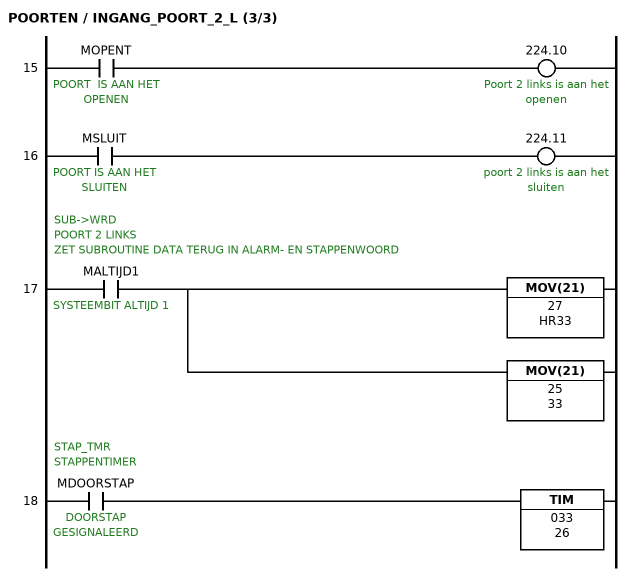
; [picture p445: POORTEN / INGANG_POORT_2_L, rungs 15-18]
; rung 15
LD MOPENT  ; POORT  IS AAN HET OPENEN
OUT 224.10  ; Poort 2 links is aan het openen
; rung 16
LD MSLUIT  ; POORT IS AAN HET SLUITEN
OUT 224.11  ; poort 2 links is aan het sluiten
; rung 17: SUB->WRD / POORT 2 LINKS / ZET SUBROUTINE DATA TERUG IN ALARM- EN STAPPENWOORD
LD MALTIJD1  ; SYSTEEMBIT ALTIJD 1
MOV(21) 27 HR33
MOV(21) 25 33
; rung 18: STAP_TMR / STAPPENTIMER
LD MDOORSTAP  ; DOORSTAP GESIGNALEERD
TIM 033 26

### Section INGANG_POORT_2_R

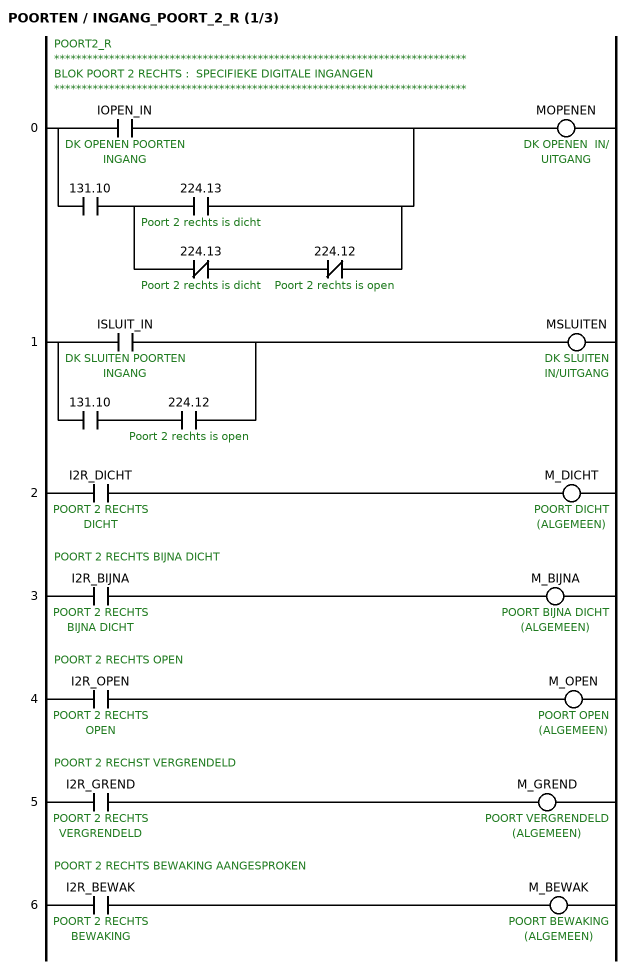
; rung 0: POORT2_R / *************************************************************************** / BLOK POORT 2 RECHTS :  SPECIFIEKE DIGITALE INGANGEN / ***************************************************************************
LD IOPEN_IN  ; DK OPENEN POORTEN INGANG
LD 131.10
LD 224.13  ; Poort 2 rechts is dicht
LDNOT 224.13  ; Poort 2 rechts is dicht
ANDNOT 224.12  ; Poort 2 rechts is open
ORLD
ANDLD
ORLD
OUT MOPENEN  ; DK OPENEN  IN/ UITGANG
; rung 1
LD ISLUIT_IN  ; DK SLUITEN POORTEN INGANG
LD 131.10
AND 224.12  ; Poort 2 rechts is open
ORLD
OUT MSLUITEN  ; DK SLUITEN  IN/UITGANG
; rung 2
LD I2R_DICHT  ; POORT 2 RECHTS DICHT
OUT M_DICHT  ; POORT DICHT (ALGEMEEN)
; rung 3: POORT 2 RECHTS BIJNA DICHT
LD I2R_BIJNA  ; POORT 2 RECHTS BIJNA DICHT
OUT M_BIJNA  ; POORT BIJNA DICHT  (ALGEMEEN)
; rung 4: POORT 2 RECHTS OPEN
LD I2R_OPEN  ; POORT 2 RECHTS OPEN
OUT M_OPEN  ; POORT OPEN (ALGEMEEN)
; rung 5: POORT 2 RECHST VERGRENDELD
LD I2R_GREND  ; POORT 2 RECHTS VERGRENDELD
OUT M_GREND  ; POORT VERGRENDELD (ALGEMEEN)
; rung 6: POORT 2 RECHTS BEWAKING AANGESPROKEN
LD I2R_BEWAK  ; POORT 2 RECHTS BEWAKING
OUT M_BEWAK  ; POORT BEWAKING (ALGEMEEN)

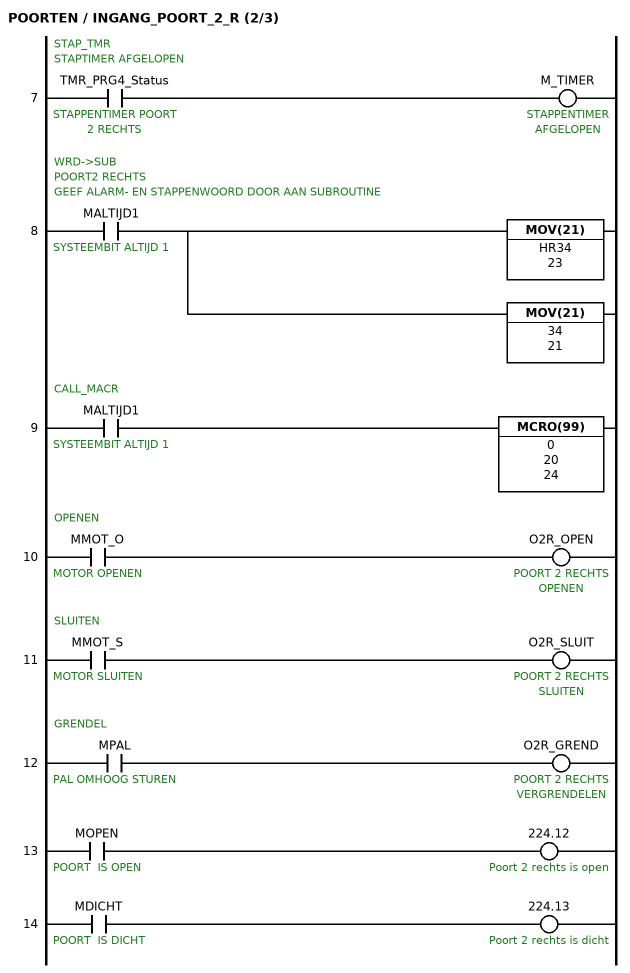
; rung 7: STAP_TMR / STAPTIMER AFGELOPEN
LD TMR_PRG4_Status  ; STAPPENTIMER POORT 2 RECHTS
OUT M_TIMER  ; STAPPENTIMER AFGELOPEN
; rung 8: WRD->SUB / POORT2 RECHTS / GEEF ALARM- EN STAPPENWOORD DOOR AAN SUBROUTINE
LD MALTIJD1  ; SYSTEEMBIT ALTIJD 1
MOV(21) HR34 23
MOV(21) 34 21
; rung 9: CALL_MACR
LD MALTIJD1  ; SYSTEEMBIT ALTIJD 1
MCRO(99) 0 20 24
; rung 10: OPENEN
LD MMOT_O  ; MOTOR OPENEN
OUT O2R_OPEN  ; POORT 2 RECHTS OPENEN
; rung 11: SLUITEN
LD MMOT_S  ; MOTOR SLUITEN
OUT O2R_SLUIT  ; POORT 2 RECHTS SLUITEN
; rung 12: GRENDEL
LD MPAL  ; PAL OMHOOG STUREN
OUT O2R_GREND  ; POORT 2 RECHTS VERGRENDELEN
; rung 13
LD MOPEN  ; POORT  IS OPEN
OUT 224.12  ; Poort 2 rechts is open
; rung 14
LD MDICHT  ; POORT  IS DICHT
OUT 224.13  ; Poort 2 rechts is dicht

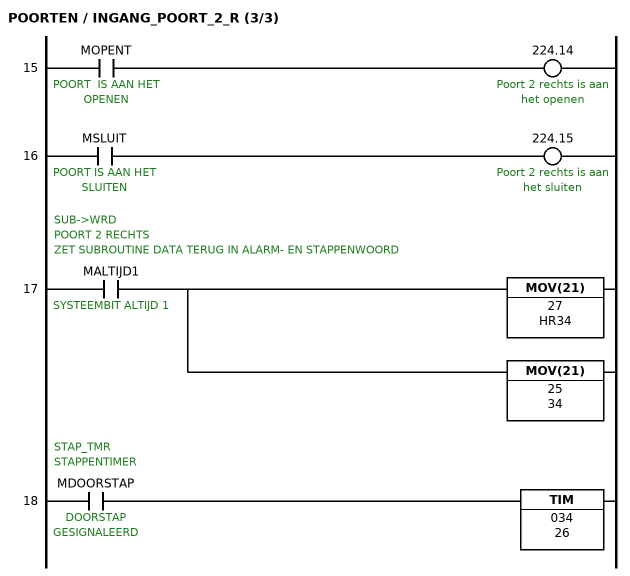
; rung 15
LD MOPENT  ; POORT  IS AAN HET OPENEN
OUT 224.14  ; Poort 2 rechts is aan het openen
; rung 16
LD MSLUIT  ; POORT IS AAN HET SLUITEN
OUT 224.15  ; Poort 2 rechts is aan het sluiten
; rung 17: SUB->WRD / POORT 2 RECHTS / ZET SUBROUTINE DATA TERUG IN ALARM- EN STAPPENWOORD
LD MALTIJD1  ; SYSTEEMBIT ALTIJD 1
MOV(21) 27 HR34
MOV(21) 25 34
; rung 18: STAP_TMR / STAPPENTIMER
LD MDOORSTAP  ; DOORSTAP GESIGNALEERD
TIM 034 26

### Section UITGANG_POORT_3_L

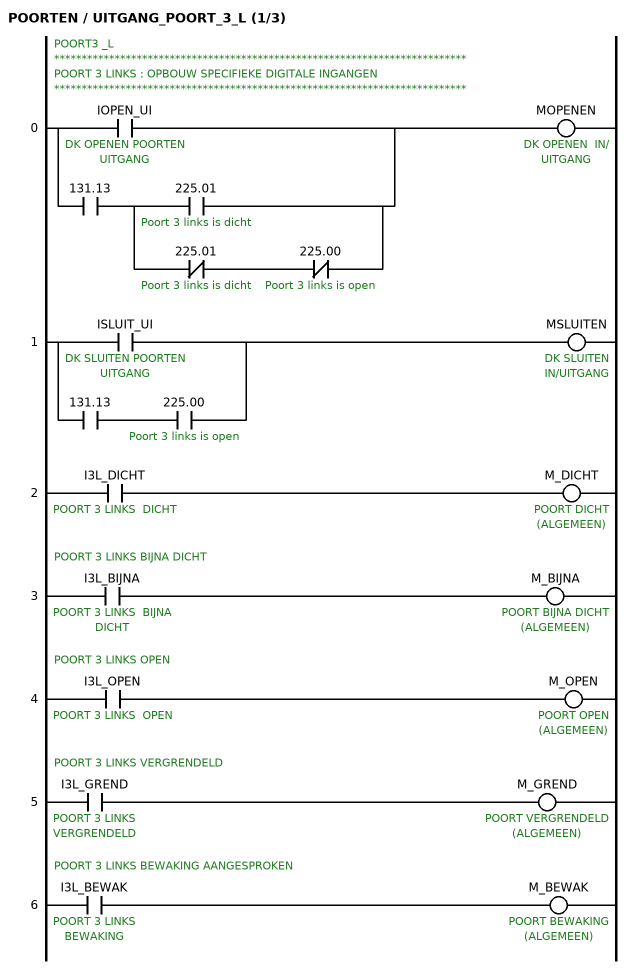
; rung 0: POORT3 _L / *************************************************************************** / POORT 3 LINKS : OPBOUW SPECIFIEKE DIGITALE INGANGEN / ***************************************************************************
LD IOPEN_UI  ; DK OPENEN POORTEN UITGANG
LD 131.13
LD 225.01  ; Poort 3 links is dicht
LDNOT 225.01  ; Poort 3 links is dicht
ANDNOT 225.00  ; Poort 3 links is open
ORLD
ANDLD
ORLD
OUT MOPENEN  ; DK OPENEN  IN/ UITGANG
; rung 1
LD ISLUIT_UI  ; DK SLUITEN POORTEN UITGANG
LD 131.13
AND 225.00  ; Poort 3 links is open
ORLD
OUT MSLUITEN  ; DK SLUITEN  IN/UITGANG
; rung 2
LD I3L_DICHT  ; POORT 3 LINKS  DICHT
OUT M_DICHT  ; POORT DICHT (ALGEMEEN)
; rung 3: POORT 3 LINKS BIJNA DICHT
LD I3L_BIJNA  ; POORT 3 LINKS  BIJNA DICHT
OUT M_BIJNA  ; POORT BIJNA DICHT  (ALGEMEEN)
; rung 4: POORT 3 LINKS OPEN
LD I3L_OPEN  ; POORT 3 LINKS  OPEN
OUT M_OPEN  ; POORT OPEN (ALGEMEEN)
; rung 5: POORT 3 LINKS VERGRENDELD
LD I3L_GREND  ; POORT 3 LINKS VERGRENDELD
OUT M_GREND  ; POORT VERGRENDELD (ALGEMEEN)
; rung 6: POORT 3 LINKS BEWAKING AANGESPROKEN
LD I3L_BEWAK  ; POORT 3 LINKS BEWAKING
OUT M_BEWAK  ; POORT BEWAKING (ALGEMEEN)

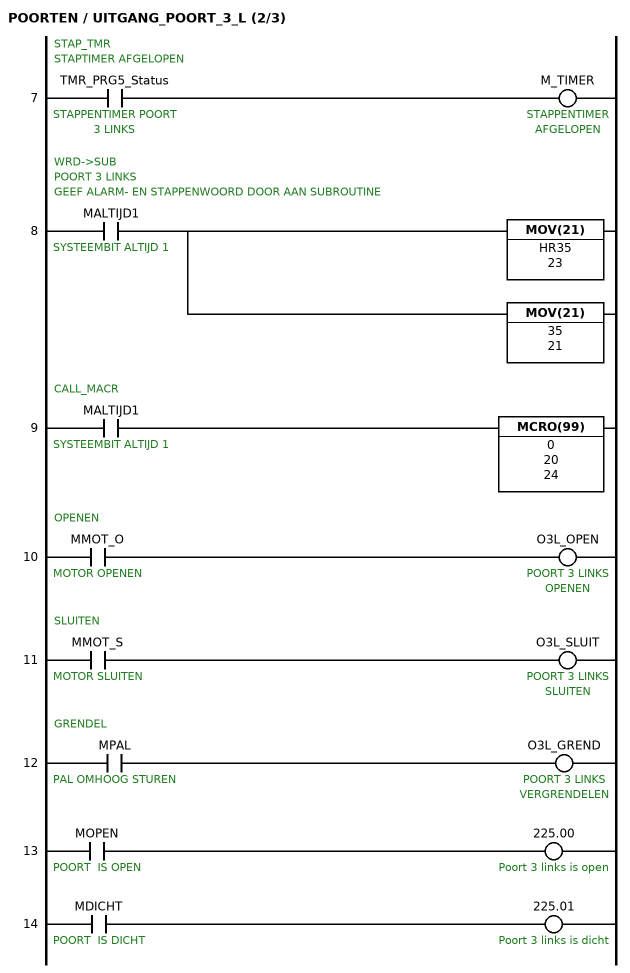
; rung 7: STAP_TMR / STAPTIMER AFGELOPEN
LD TMR_PRG5_Status  ; STAPPENTIMER POORT 3 LINKS
OUT M_TIMER  ; STAPPENTIMER AFGELOPEN
; rung 8: WRD->SUB / POORT 3 LINKS / GEEF ALARM- EN STAPPENWOORD DOOR AAN SUBROUTINE
LD MALTIJD1  ; SYSTEEMBIT ALTIJD 1
MOV(21) HR35 23
MOV(21) 35 21
; rung 9: CALL_MACR
LD MALTIJD1  ; SYSTEEMBIT ALTIJD 1
MCRO(99) 0 20 24
; rung 10: OPENEN
LD MMOT_O  ; MOTOR OPENEN
OUT O3L_OPEN  ; POORT 3 LINKS OPENEN
; rung 11: SLUITEN
LD MMOT_S  ; MOTOR SLUITEN
OUT O3L_SLUIT  ; POORT 3 LINKS SLUITEN
; rung 12: GRENDEL
LD MPAL  ; PAL OMHOOG STUREN
OUT O3L_GREND  ; POORT 3 LINKS VERGRENDELEN
; rung 13
LD MOPEN  ; POORT  IS OPEN
OUT 225.00  ; Poort 3 links is open
; rung 14
LD MDICHT  ; POORT  IS DICHT
OUT 225.01  ; Poort 3 links is dicht

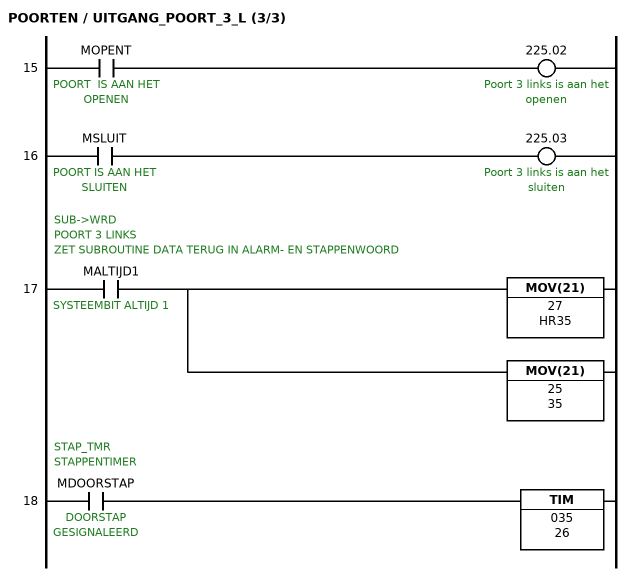
; rung 15
LD MOPENT  ; POORT  IS AAN HET OPENEN
OUT 225.02  ; Poort 3 links is aan het openen
; rung 16
LD MSLUIT  ; POORT IS AAN HET SLUITEN
OUT 225.03  ; Poort 3 links is aan het sluiten
; rung 17: SUB->WRD / POORT 3 LINKS / ZET SUBROUTINE DATA TERUG IN ALARM- EN STAPPENWOORD
LD MALTIJD1  ; SYSTEEMBIT ALTIJD 1
MOV(21) 27 HR35
MOV(21) 25 35
; rung 18: STAP_TMR / STAPPENTIMER
LD MDOORSTAP  ; DOORSTAP GESIGNALEERD
TIM 035 26

### Section UITGANG_POORT_3_R

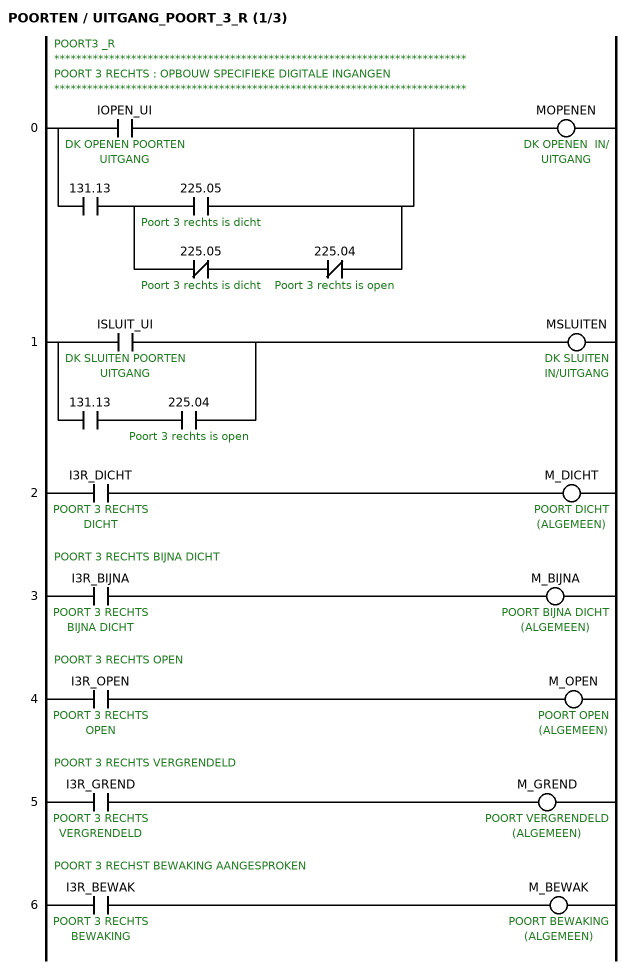
; rung 0: POORT3 _R / *************************************************************************** / POORT 3 RECHTS : OPBOUW SPECIFIEKE DIGITALE INGANGEN / ***************************************************************************
LD IOPEN_UI  ; DK OPENEN POORTEN UITGANG
LD 131.13
LD 225.05  ; Poort 3 rechts is dicht
LDNOT 225.05  ; Poort 3 rechts is dicht
ANDNOT 225.04  ; Poort 3 rechts is open
ORLD
ANDLD
ORLD
OUT MOPENEN  ; DK OPENEN  IN/ UITGANG
; rung 1
LD ISLUIT_UI  ; DK SLUITEN POORTEN UITGANG
LD 131.13
AND 225.04  ; Poort 3 rechts is open
ORLD
OUT MSLUITEN  ; DK SLUITEN  IN/UITGANG
; rung 2
LD I3R_DICHT  ; POORT 3 RECHTS DICHT
OUT M_DICHT  ; POORT DICHT (ALGEMEEN)
; rung 3: POORT 3 RECHTS BIJNA DICHT
LD I3R_BIJNA  ; POORT 3 RECHTS BIJNA DICHT
OUT M_BIJNA  ; POORT BIJNA DICHT  (ALGEMEEN)
; rung 4: POORT 3 RECHTS OPEN
LD I3R_OPEN  ; POORT 3 RECHTS OPEN
OUT M_OPEN  ; POORT OPEN (ALGEMEEN)
; rung 5: POORT 3 RECHTS VERGRENDELD
LD I3R_GREND  ; POORT 3 RECHTS VERGRENDELD
OUT M_GREND  ; POORT VERGRENDELD (ALGEMEEN)
; rung 6: POORT 3 RECHST BEWAKING AANGESPROKEN
LD I3R_BEWAK  ; POORT 3 RECHTS BEWAKING
OUT M_BEWAK  ; POORT BEWAKING (ALGEMEEN)

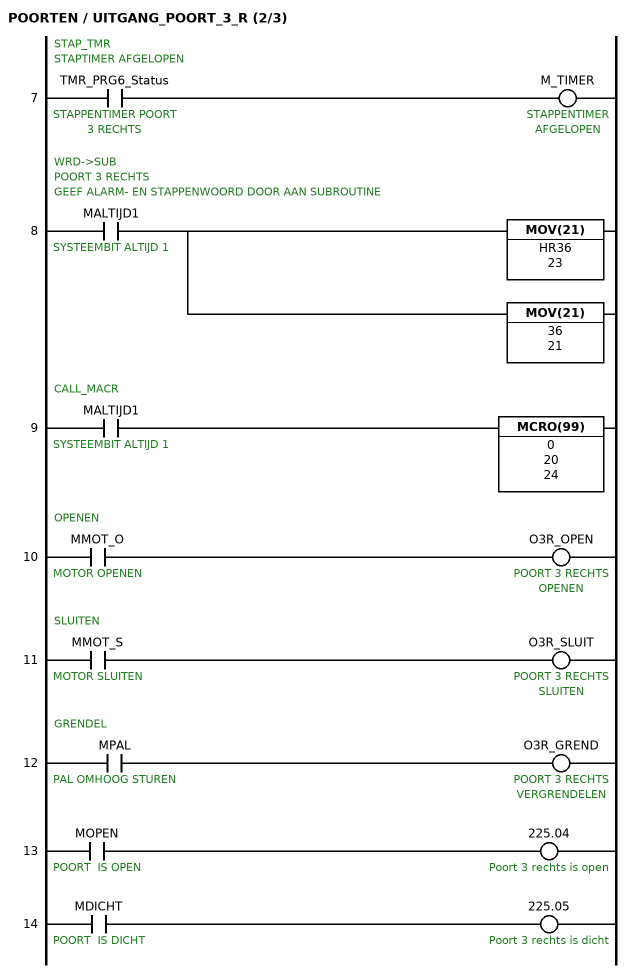
; rung 7: STAP_TMR / STAPTIMER AFGELOPEN
LD TMR_PRG6_Status  ; STAPPENTIMER POORT 3 RECHTS
OUT M_TIMER  ; STAPPENTIMER AFGELOPEN
; rung 8: WRD->SUB / POORT 3 RECHTS / GEEF ALARM- EN STAPPENWOORD DOOR AAN SUBROUTINE
LD MALTIJD1  ; SYSTEEMBIT ALTIJD 1
MOV(21) HR36 23
MOV(21) 36 21
; rung 9: CALL_MACR
LD MALTIJD1  ; SYSTEEMBIT ALTIJD 1
MCRO(99) 0 20 24
; rung 10: OPENEN
LD MMOT_O  ; MOTOR OPENEN
OUT O3R_OPEN  ; POORT 3 RECHTS OPENEN
; rung 11: SLUITEN
LD MMOT_S  ; MOTOR SLUITEN
OUT O3R_SLUIT  ; POORT 3 RECHTS SLUITEN
; rung 12: GRENDEL
LD MPAL  ; PAL OMHOOG STUREN
OUT O3R_GREND  ; POORT 3 RECHTS VERGRENDELEN
; rung 13
LD MOPEN  ; POORT  IS OPEN
OUT 225.04  ; Poort 3 rechts is open
; rung 14
LD MDICHT  ; POORT  IS DICHT
OUT 225.05  ; Poort 3 rechts is dicht

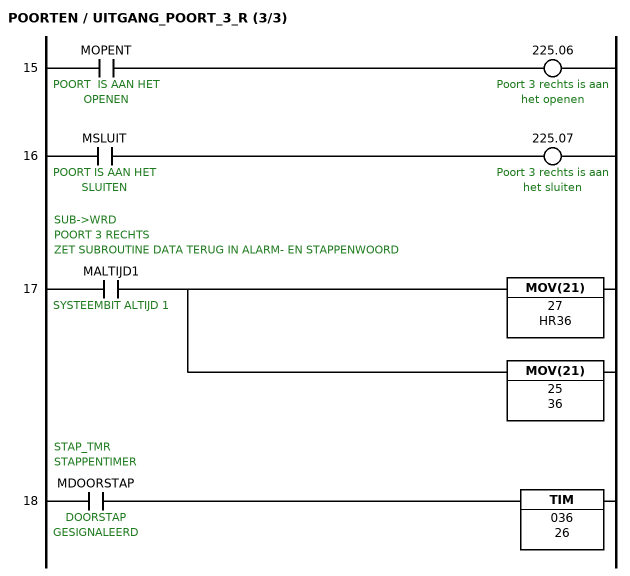
; rung 15
LD MOPENT  ; POORT  IS AAN HET OPENEN
OUT 225.06  ; Poort 3 rechts is aan het openen
; rung 16
LD MSLUIT  ; POORT IS AAN HET SLUITEN
OUT 225.07  ; Poort 3 rechts is aan het sluiten
; rung 17: SUB->WRD / POORT 3 RECHTS / ZET SUBROUTINE DATA TERUG IN ALARM- EN STAPPENWOORD
LD MALTIJD1  ; SYSTEEMBIT ALTIJD 1
MOV(21) 27 HR36
MOV(21) 25 36
; rung 18: STAP_TMR / STAPPENTIMER
LD MDOORSTAP  ; DOORSTAP GESIGNALEERD
TIM 036 26

### Section UITGANG_POORT_4_L

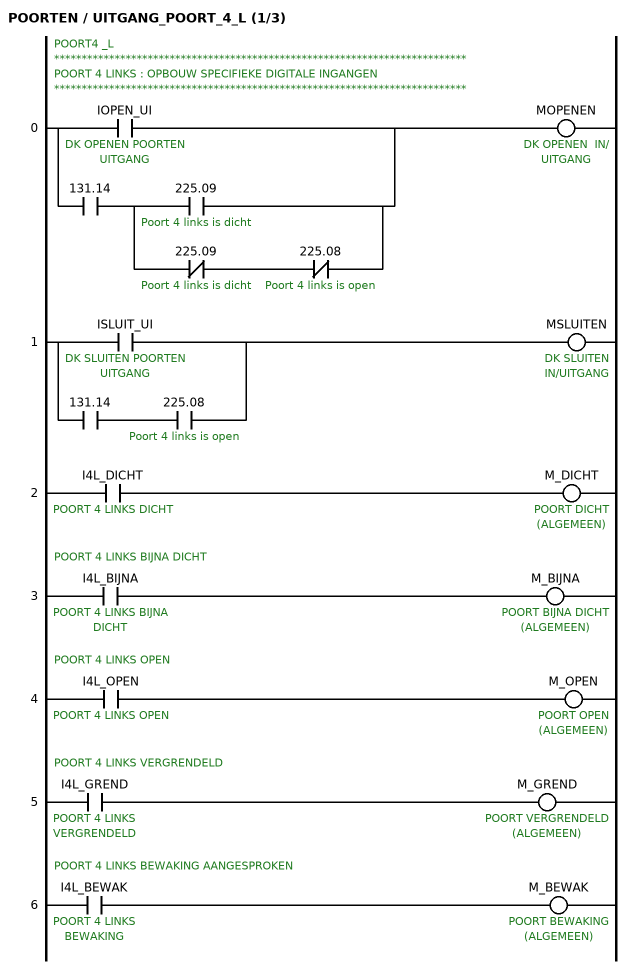
; rung 0: POORT4 _L / *************************************************************************** / POORT 4 LINKS : OPBOUW SPECIFIEKE DIGITALE INGANGEN / ***************************************************************************
LD IOPEN_UI  ; DK OPENEN POORTEN UITGANG
LD 131.14
LD 225.09  ; Poort 4 links is dicht
LDNOT 225.09  ; Poort 4 links is dicht
ANDNOT 225.08  ; Poort 4 links is open
ORLD
ANDLD
ORLD
OUT MOPENEN  ; DK OPENEN  IN/ UITGANG
; rung 1
LD ISLUIT_UI  ; DK SLUITEN POORTEN UITGANG
LD 131.14
AND 225.08  ; Poort 4 links is open
ORLD
OUT MSLUITEN  ; DK SLUITEN  IN/UITGANG
; rung 2
LD I4L_DICHT  ; POORT 4 LINKS DICHT
OUT M_DICHT  ; POORT DICHT (ALGEMEEN)
; rung 3: POORT 4 LINKS BIJNA DICHT
LD I4L_BIJNA  ; POORT 4 LINKS BIJNA DICHT
OUT M_BIJNA  ; POORT BIJNA DICHT  (ALGEMEEN)
; rung 4: POORT 4 LINKS OPEN
LD I4L_OPEN  ; POORT 4 LINKS OPEN
OUT M_OPEN  ; POORT OPEN (ALGEMEEN)
; rung 5: POORT 4 LINKS VERGRENDELD
LD I4L_GREND  ; POORT 4 LINKS VERGRENDELD
OUT M_GREND  ; POORT VERGRENDELD (ALGEMEEN)
; rung 6: POORT 4 LINKS BEWAKING AANGESPROKEN
LD I4L_BEWAK  ; POORT 4 LINKS BEWAKING
OUT M_BEWAK  ; POORT BEWAKING (ALGEMEEN)

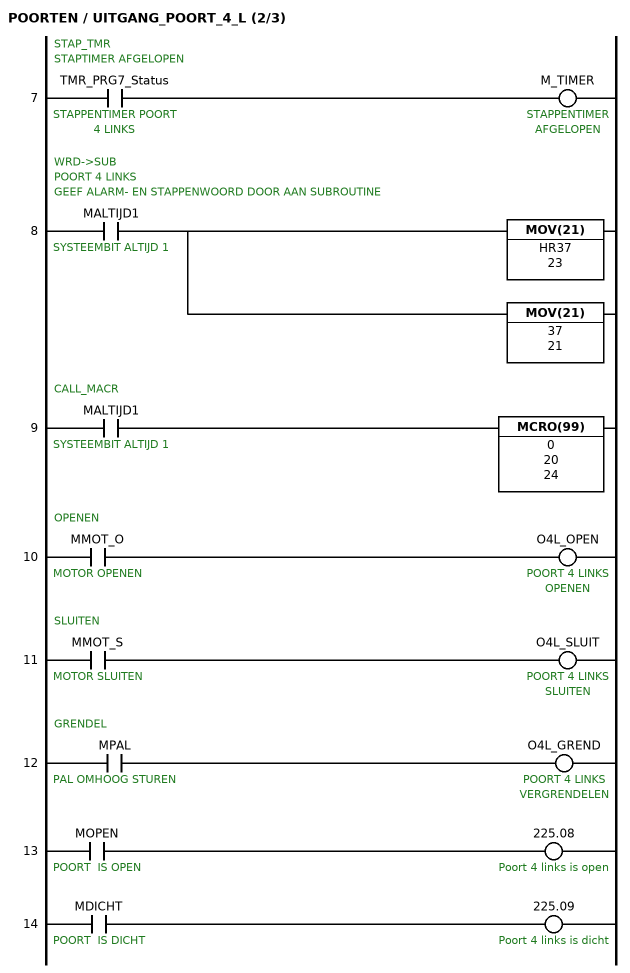
; rung 7: STAP_TMR / STAPTIMER AFGELOPEN
LD TMR_PRG7_Status  ; STAPPENTIMER POORT 4 LINKS
OUT M_TIMER  ; STAPPENTIMER AFGELOPEN
; rung 8: WRD->SUB / POORT 4 LINKS / GEEF ALARM- EN STAPPENWOORD DOOR AAN SUBROUTINE
LD MALTIJD1  ; SYSTEEMBIT ALTIJD 1
MOV(21) HR37 23
MOV(21) 37 21
; rung 9: CALL_MACR
LD MALTIJD1  ; SYSTEEMBIT ALTIJD 1
MCRO(99) 0 20 24
; rung 10: OPENEN
LD MMOT_O  ; MOTOR OPENEN
OUT O4L_OPEN  ; POORT 4 LINKS OPENEN
; rung 11: SLUITEN
LD MMOT_S  ; MOTOR SLUITEN
OUT O4L_SLUIT  ; POORT 4 LINKS SLUITEN
; rung 12: GRENDEL
LD MPAL  ; PAL OMHOOG STUREN
OUT O4L_GREND  ; POORT 4 LINKS VERGRENDELEN
; rung 13
LD MOPEN  ; POORT  IS OPEN
OUT 225.08  ; Poort 4 links is open
; rung 14
LD MDICHT  ; POORT  IS DICHT
OUT 225.09  ; Poort 4 links is dicht

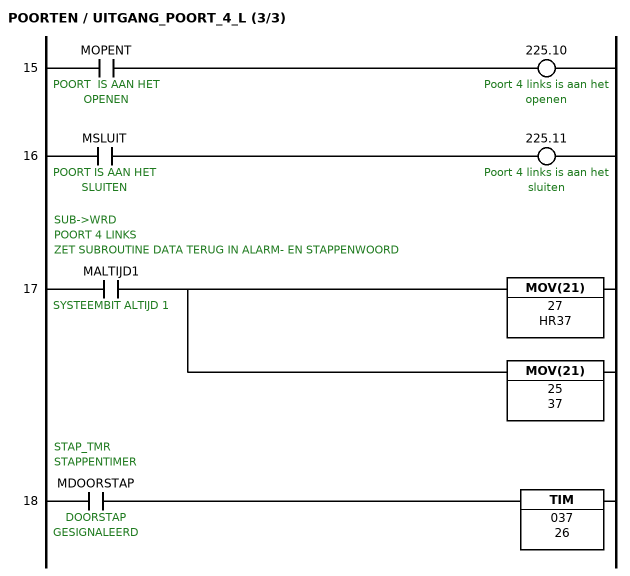
; rung 15
LD MOPENT  ; POORT  IS AAN HET OPENEN
OUT 225.10  ; Poort 4 links is aan het openen
; rung 16
LD MSLUIT  ; POORT IS AAN HET SLUITEN
OUT 225.11  ; Poort 4 links is aan het sluiten
; rung 17: SUB->WRD / POORT 4 LINKS / ZET SUBROUTINE DATA TERUG IN ALARM- EN STAPPENWOORD
LD MALTIJD1  ; SYSTEEMBIT ALTIJD 1
MOV(21) 27 HR37
MOV(21) 25 37
; rung 18: STAP_TMR / STAPPENTIMER
LD MDOORSTAP  ; DOORSTAP GESIGNALEERD
TIM 037 26

### Section UITGANG_POORT_4_R

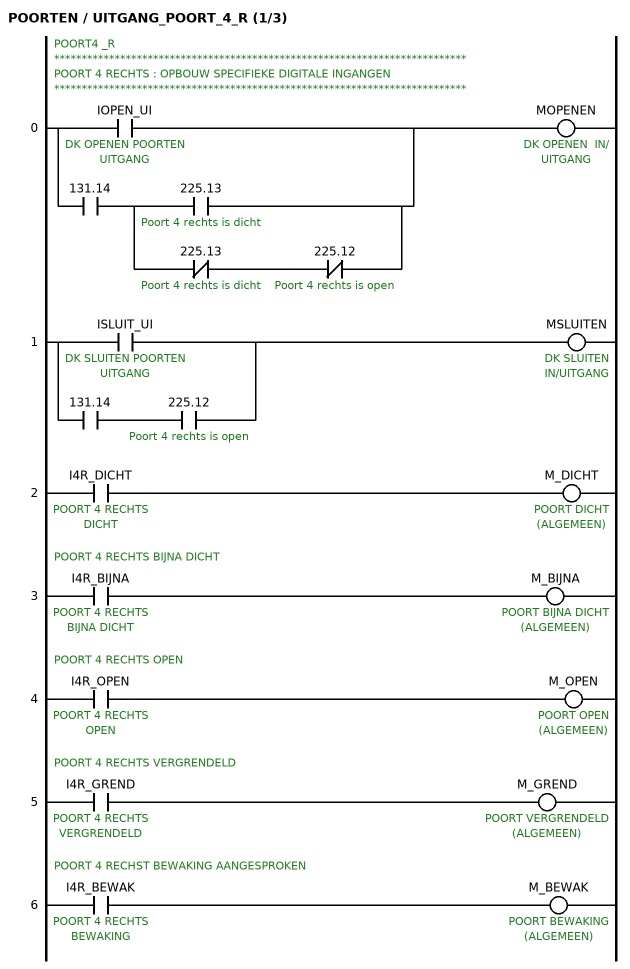
; rung 0: POORT4 _R / *************************************************************************** / POORT 4 RECHTS : OPBOUW SPECIFIEKE DIGITALE INGANGEN / ***************************************************************************
LD IOPEN_UI  ; DK OPENEN POORTEN UITGANG
LD 131.14
LD 225.13  ; Poort 4 rechts is dicht
LDNOT 225.13  ; Poort 4 rechts is dicht
ANDNOT 225.12  ; Poort 4 rechts is open
ORLD
ANDLD
ORLD
OUT MOPENEN  ; DK OPENEN  IN/ UITGANG
; rung 1
LD ISLUIT_UI  ; DK SLUITEN POORTEN UITGANG
LD 131.14
AND 225.12  ; Poort 4 rechts is open
ORLD
OUT MSLUITEN  ; DK SLUITEN  IN/UITGANG
; rung 2
LD I4R_DICHT  ; POORT 4 RECHTS DICHT
OUT M_DICHT  ; POORT DICHT (ALGEMEEN)
; rung 3: POORT 4 RECHTS BIJNA DICHT
LD I4R_BIJNA  ; POORT 4 RECHTS BIJNA DICHT
OUT M_BIJNA  ; POORT BIJNA DICHT  (ALGEMEEN)
; rung 4: POORT 4 RECHTS OPEN
LD I4R_OPEN  ; POORT 4 RECHTS OPEN
OUT M_OPEN  ; POORT OPEN (ALGEMEEN)
; rung 5: POORT 4 RECHTS VERGRENDELD
LD I4R_GREND  ; POORT 4 RECHTS VERGRENDELD
OUT M_GREND  ; POORT VERGRENDELD (ALGEMEEN)
; rung 6: POORT 4 RECHST BEWAKING AANGESPROKEN
LD I4R_BEWAK  ; POORT 4 RECHTS BEWAKING
OUT M_BEWAK  ; POORT BEWAKING (ALGEMEEN)

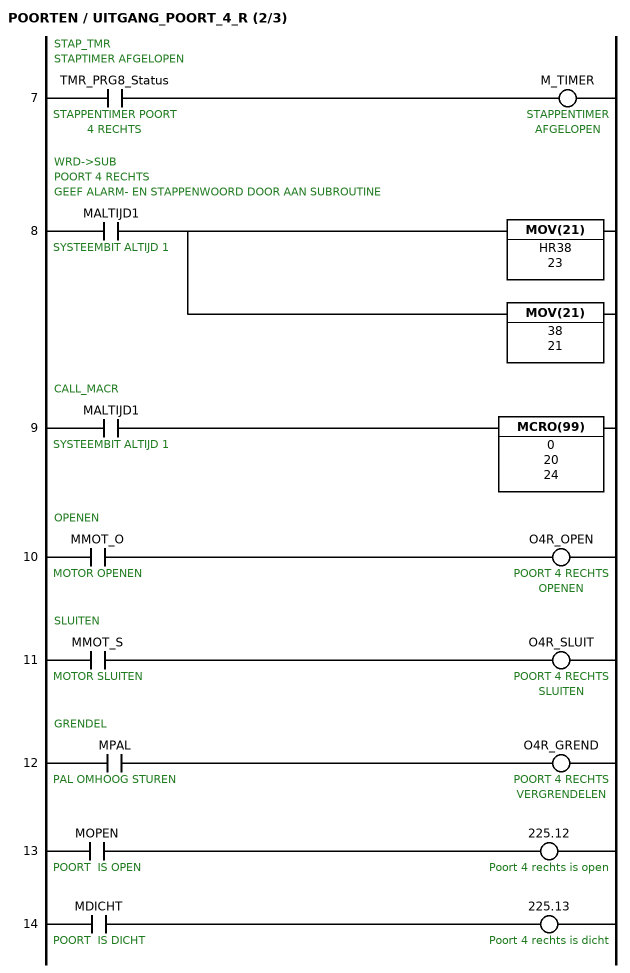
; rung 7: STAP_TMR / STAPTIMER AFGELOPEN
LD TMR_PRG8_Status  ; STAPPENTIMER POORT 4 RECHTS
OUT M_TIMER  ; STAPPENTIMER AFGELOPEN
; rung 8: WRD->SUB / POORT 4 RECHTS / GEEF ALARM- EN STAPPENWOORD DOOR AAN SUBROUTINE
LD MALTIJD1  ; SYSTEEMBIT ALTIJD 1
MOV(21) HR38 23
MOV(21) 38 21
; rung 9: CALL_MACR
LD MALTIJD1  ; SYSTEEMBIT ALTIJD 1
MCRO(99) 0 20 24
; rung 10: OPENEN
LD MMOT_O  ; MOTOR OPENEN
OUT O4R_OPEN  ; POORT 4 RECHTS OPENEN
; rung 11: SLUITEN
LD MMOT_S  ; MOTOR SLUITEN
OUT O4R_SLUIT  ; POORT 4 RECHTS SLUITEN
; rung 12: GRENDEL
LD MPAL  ; PAL OMHOOG STUREN
OUT O4R_GREND  ; POORT 4 RECHTS VERGRENDELEN
; rung 13
LD MOPEN  ; POORT  IS OPEN
OUT 225.12  ; Poort 4 rechts is open
; rung 14
LD MDICHT  ; POORT  IS DICHT
OUT 225.13  ; Poort 4 rechts is dicht

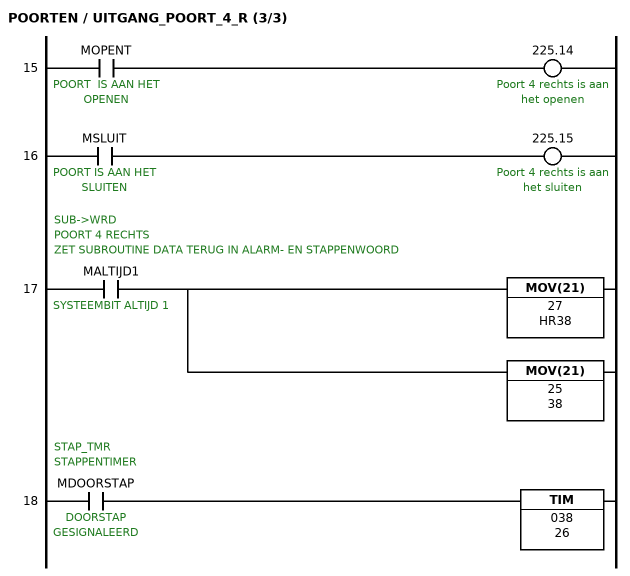
; rung 15
LD MOPENT  ; POORT  IS AAN HET OPENEN
OUT 225.14  ; Poort 4 rechts is aan het openen
; rung 16
LD MSLUIT  ; POORT IS AAN HET SLUITEN
OUT 225.15  ; Poort 4 rechts is aan het sluiten
; rung 17: SUB->WRD / POORT 4 RECHTS / ZET SUBROUTINE DATA TERUG IN ALARM- EN STAPPENWOORD
LD MALTIJD1  ; SYSTEEMBIT ALTIJD 1
MOV(21) 27 HR38
MOV(21) 25 38
; rung 18: STAP_TMR / STAPPENTIMER
LD MDOORSTAP  ; DOORSTAP GESIGNALEERD
TIM 038 26

### Section POORTEN_ALL
; POORTEN_ALL

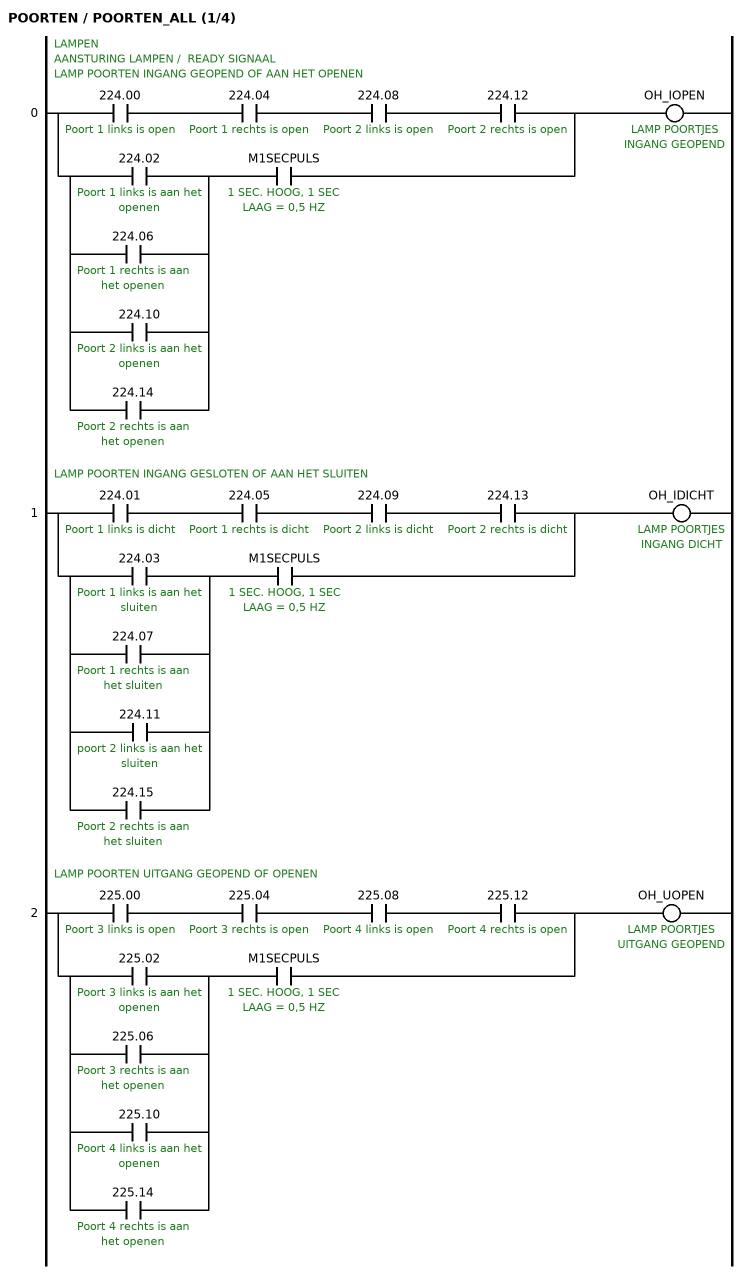
; rung 0: LAMPEN / AANSTURING LAMPEN /  READY SIGNAAL / LAMP POORTEN INGANG GEOPEND OF AAN HET OPENEN
LD 224.00  ; Poort 1 links is open
AND 224.04  ; Poort 1 rechts is open
AND 224.08  ; Poort 2 links is open
AND 224.12  ; Poort 2 rechts is open
LD 224.02  ; Poort 1 links is aan het openen
OR 224.06  ; Poort 1 rechts is aan het openen
OR 224.10  ; Poort 2 links is aan het openen
OR 224.14  ; Poort 2 rechts is aan het openen
AND M1SECPULS  ; 1 SEC. HOOG, 1 SEC LAAG = 0,5 HZ
ORLD
OUT OH_IOPEN  ; LAMP POORTJES INGANG GEOPEND
; rung 1: LAMP POORTEN INGANG GESLOTEN OF AAN HET SLUITEN
LD 224.01  ; Poort 1 links is dicht
AND 224.05  ; Poort 1 rechts is dicht
AND 224.09  ; Poort 2 links is dicht
AND 224.13  ; Poort 2 rechts is dicht
LD 224.03  ; Poort 1 links is aan het sluiten
OR 224.07  ; Poort 1 rechts is aan het sluiten
OR 224.11  ; poort 2 links is aan het sluiten
OR 224.15  ; Poort 2 rechts is aan het sluiten
AND M1SECPULS  ; 1 SEC. HOOG, 1 SEC LAAG = 0,5 HZ
ORLD
OUT OH_IDICHT  ; LAMP POORTJES INGANG DICHT
; rung 2: LAMP POORTEN UITGANG GEOPEND OF OPENEN
LD 225.00  ; Poort 3 links is open
AND 225.04  ; Poort 3 rechts is open
AND 225.08  ; Poort 4 links is open
AND 225.12  ; Poort 4 rechts is open
LD 225.02  ; Poort 3 links is aan het openen
OR 225.06  ; Poort 3 rechts is aan het openen
OR 225.10  ; Poort 4 links is aan het openen
OR 225.14  ; Poort 4 rechts is aan het openen
AND M1SECPULS  ; 1 SEC. HOOG, 1 SEC LAAG = 0,5 HZ
ORLD
OUT OH_UOPEN  ; LAMP POORTJES UITGANG GEOPEND

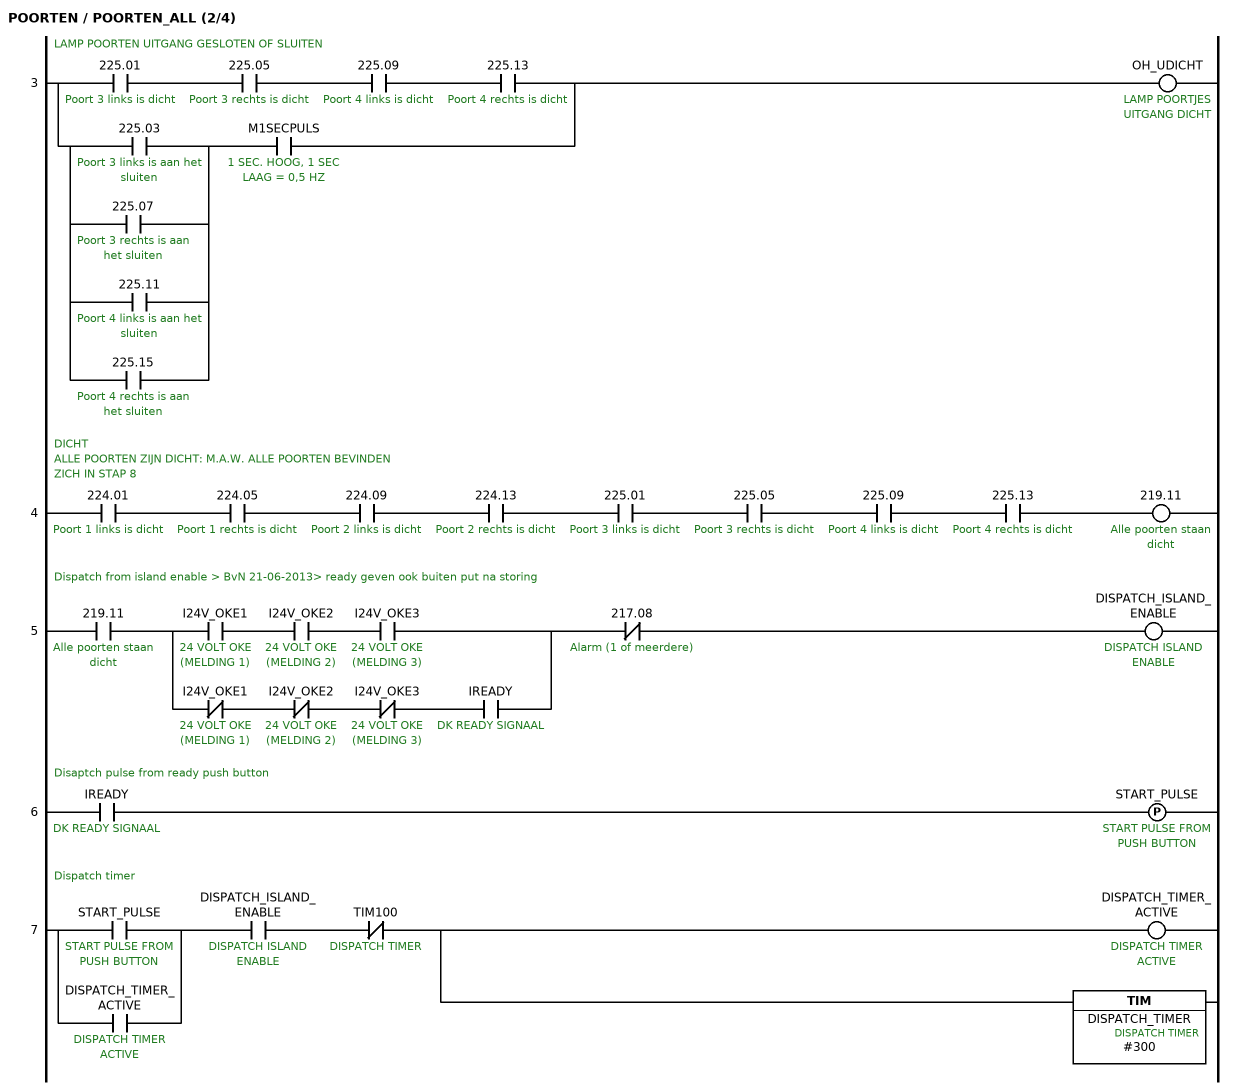
; rung 3: LAMP POORTEN UITGANG GESLOTEN OF SLUITEN
LD 225.01  ; Poort 3 links is dicht
AND 225.05  ; Poort 3 rechts is dicht
AND 225.09  ; Poort 4 links is dicht
AND 225.13  ; Poort 4 rechts is dicht
LD 225.03  ; Poort 3 links is aan het sluiten
OR 225.07  ; Poort 3 rechts is aan het sluiten
OR 225.11  ; Poort 4 links is aan het sluiten
OR 225.15  ; Poort 4 rechts is aan het sluiten
AND M1SECPULS  ; 1 SEC. HOOG, 1 SEC LAAG = 0,5 HZ
ORLD
OUT OH_UDICHT  ; LAMP POORTJES UITGANG DICHT
; rung 4: DICHT / ALLE POORTEN ZIJN DICHT: M.A.W. ALLE POORTEN BEVINDEN / ZICH IN STAP 8
LD 224.01  ; Poort 1 links is dicht
AND 224.05  ; Poort 1 rechts is dicht
AND 224.09  ; Poort 2 links is dicht
AND 224.13  ; Poort 2 rechts is dicht
AND 225.01  ; Poort 3 links is dicht
AND 225.05  ; Poort 3 rechts is dicht
AND 225.09  ; Poort 4 links is dicht
AND 225.13  ; Poort 4 rechts is dicht
OUT 219.11  ; Alle poorten staan dicht
; rung 5: Dispatch from island enable > BvN 21-06-2013> ready geven ook buiten put na storing
LD 219.11  ; Alle poorten staan dicht
LD I24V_OKE1  ; 24 VOLT OKE (MELDING 1)
AND I24V_OKE2  ; 24 VOLT OKE (MELDING 2)
AND I24V_OKE3  ; 24 VOLT OKE (MELDING 3)
LDNOT I24V_OKE1  ; 24 VOLT OKE (MELDING 1)
ANDNOT I24V_OKE2  ; 24 VOLT OKE (MELDING 2)
ANDNOT I24V_OKE3  ; 24 VOLT OKE (MELDING 3)
AND IREADY  ; DK READY SIGNAAL
ORLD
ANDLD
ANDNOT 217.08  ; Alarm (1 of meerdere)
OUT DISPATCH_ISLAND_ENABLE  ; DISPATCH ISLAND ENABLE
; rung 6: Disaptch pulse from ready push button
LD IREADY  ; DK READY SIGNAAL
DIFU(13) START_PULSE  ; START PULSE FROM PUSH BUTTON
; rung 7: Dispatch timer
LD START_PULSE  ; START PULSE FROM PUSH BUTTON
OR DISPATCH_TIMER_ACTIVE  ; DISPATCH TIMER ACTIVE
AND DISPATCH_ISLAND_ENABLE  ; DISPATCH ISLAND ENABLE
ANDNOT TIM100  ; DISPATCH TIMER
OUT DISPATCH_TIMER_ACTIVE  ; DISPATCH TIMER ACTIVE
TIM DISPATCH_TIMER #300  ; DISPATCH TIMER

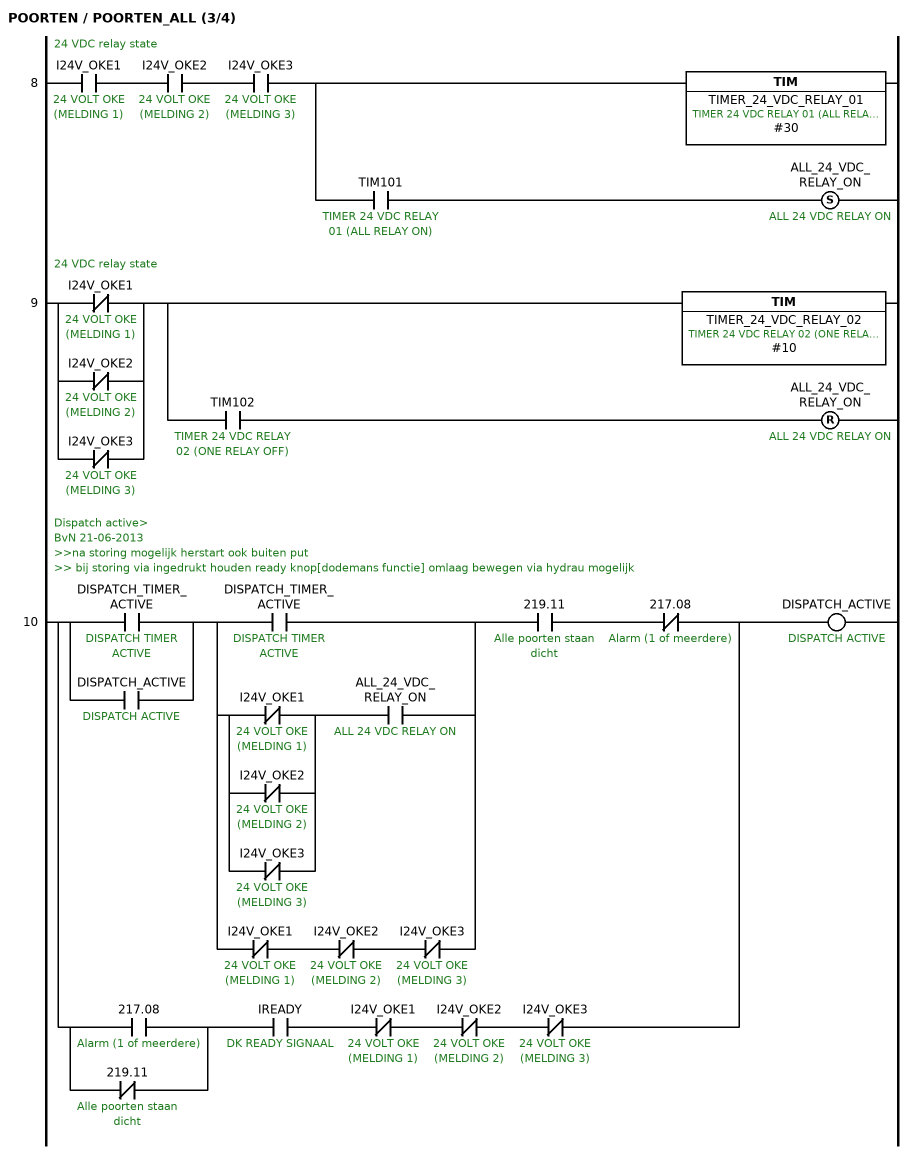
; rung 8: 24 VDC relay state
LD I24V_OKE1  ; 24 VOLT OKE (MELDING 1)
AND I24V_OKE2  ; 24 VOLT OKE (MELDING 2)
AND I24V_OKE3  ; 24 VOLT OKE (MELDING 3)
TIM TIMER_24_VDC_RELAY_01 #30  ; TIMER 24 VDC RELAY 01 (ALL RELAY ON)
AND TIM101  ; TIMER 24 VDC RELAY 01 (ALL RELAY ON)
SET ALL_24_VDC_RELAY_ON  ; ALL 24 VDC RELAY ON
; rung 9: 24 VDC relay state
LDNOT I24V_OKE1  ; 24 VOLT OKE (MELDING 1)
ORNOT I24V_OKE2  ; 24 VOLT OKE (MELDING 2)
ORNOT I24V_OKE3  ; 24 VOLT OKE (MELDING 3)
TIM TIMER_24_VDC_RELAY_02 #10  ; TIMER 24 VDC RELAY 02 (ONE RELAY OFF)
AND TIM102  ; TIMER 24 VDC RELAY 02 (ONE RELAY OFF)
RSET ALL_24_VDC_RELAY_ON  ; ALL 24 VDC RELAY ON
; rung 10: Dispatch active> / BvN 21-06-2013 / >>na storing mogelijk herstart ook buiten put / >> bij storing via ingedrukt houden ready knop[dodemans functie] omlaag bewegen via hydrau mogelijk
LD DISPATCH_TIMER_ACTIVE  ; DISPATCH TIMER ACTIVE
OR DISPATCH_ACTIVE  ; DISPATCH ACTIVE
LD DISPATCH_TIMER_ACTIVE  ; DISPATCH TIMER ACTIVE
LDNOT I24V_OKE1  ; 24 VOLT OKE (MELDING 1)
ORNOT I24V_OKE2  ; 24 VOLT OKE (MELDING 2)
ORNOT I24V_OKE3  ; 24 VOLT OKE (MELDING 3)
AND ALL_24_VDC_RELAY_ON  ; ALL 24 VDC RELAY ON
ORLD
LDNOT I24V_OKE1  ; 24 VOLT OKE (MELDING 1)
ANDNOT I24V_OKE2  ; 24 VOLT OKE (MELDING 2)
ANDNOT I24V_OKE3  ; 24 VOLT OKE (MELDING 3)
ORLD
ANDLD
AND 219.11  ; Alle poorten staan dicht
ANDNOT 217.08  ; Alarm (1 of meerdere)
LD 217.08  ; Alarm (1 of meerdere)
ORNOT 219.11  ; Alle poorten staan dicht
AND IREADY  ; DK READY SIGNAAL
ANDNOT I24V_OKE1  ; 24 VOLT OKE (MELDING 1)
ANDNOT I24V_OKE2  ; 24 VOLT OKE (MELDING 2)
ANDNOT I24V_OKE3  ; 24 VOLT OKE (MELDING 3)
ORLD
OUT DISPATCH_ACTIVE  ; DISPATCH ACTIVE

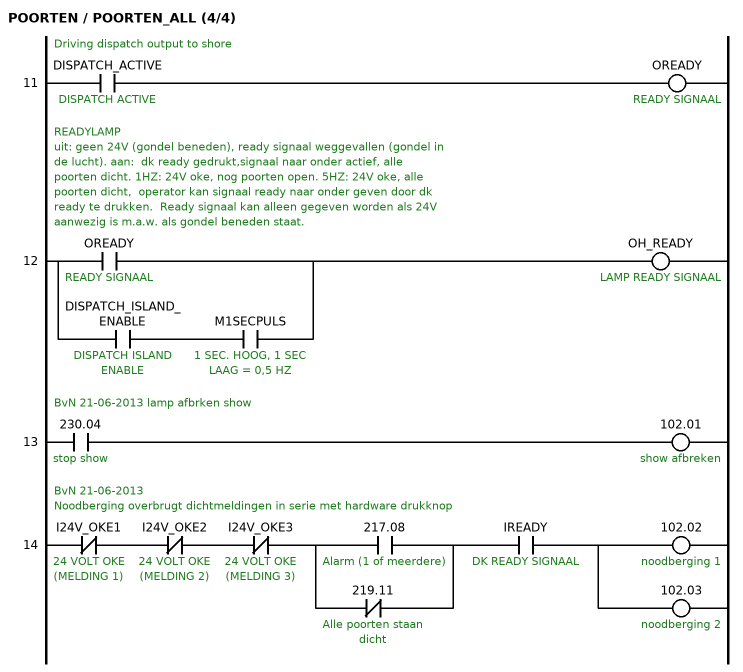
; rung 11: Driving dispatch output to shore
LD DISPATCH_ACTIVE  ; DISPATCH ACTIVE
OUT OREADY  ; READY SIGNAAL
; rung 12: READYLAMP / uit: geen 24V (gondel beneden), ready signaal weggevallen (gondel in / de lucht). aan:  dk ready gedrukt,signaal naar onder actief, alle / poorten dicht. 1HZ: 24V oke, nog poorten open. 5HZ: 24V oke, alle / poorten dicht,  operator kan signaal ready naar onder geven door dk / ready te drukken.  Ready signaal kan alleen gegeven worden als 24V / aanwezig is m.a.w. als gondel beneden staat.
LD OREADY  ; READY SIGNAAL
LD DISPATCH_ISLAND_ENABLE  ; DISPATCH ISLAND ENABLE
AND M1SECPULS  ; 1 SEC. HOOG, 1 SEC LAAG = 0,5 HZ
ORLD
OUT OH_READY  ; LAMP READY SIGNAAL
; rung 13: BvN 21-06-2013 lamp afbrken show
LD 230.04  ; stop show
OUT 102.01  ; show afbreken
; rung 14: BvN 21-06-2013 / Noodberging overbrugt dichtmeldingen in serie met hardware drukknop
LDNOT I24V_OKE1  ; 24 VOLT OKE (MELDING 1)
ANDNOT I24V_OKE2  ; 24 VOLT OKE (MELDING 2)
ANDNOT I24V_OKE3  ; 24 VOLT OKE (MELDING 3)
LD 217.08  ; Alarm (1 of meerdere)
ORNOT 219.11  ; Alle poorten staan dicht
ANDLD
AND IREADY  ; DK READY SIGNAAL
OUT 102.02  ; noodberging 1
OUT 102.03  ; noodberging 2

### Section SHOW_VERLICHTING

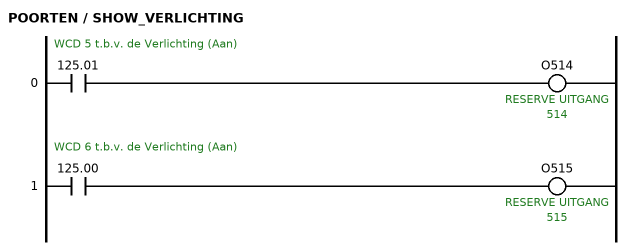
; rung 0: WCD 5 t.b.v. de Verlichting (Aan)
LD 125.01
OUT O514  ; RESERVE UITGANG 514
; rung 1: WCD 6 t.b.v. de Verlichting (Aan)
LD 125.00
OUT O515  ; RESERVE UITGANG 515

### Section MACRO_STAP

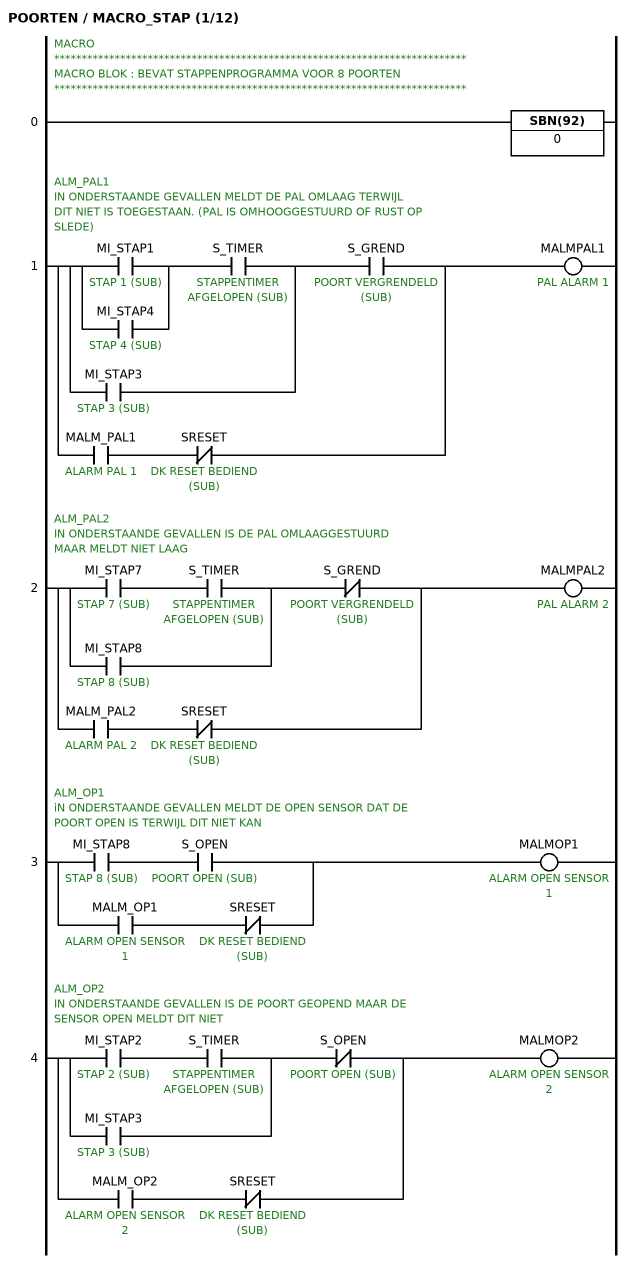
; rung 0: MACRO / *************************************************************************** / MACRO BLOK : BEVAT STAPPENPROGRAMMA VOOR 8 POORTEN / ***************************************************************************
SBN(92) 0
; rung 1: ALM_PAL1 / IN ONDERSTAANDE GEVALLEN MELDT DE PAL OMLAAG TERWIJL / DIT NIET IS TOEGESTAAN. (PAL IS OMHOOGGESTUURD OF RUST OP / SLEDE)
LD MI_STAP1  ; STAP 1 (SUB)
OR MI_STAP4  ; STAP 4 (SUB)
AND S_TIMER  ; STAPPENTIMER AFGELOPEN (SUB)
OR MI_STAP3  ; STAP 3 (SUB)
AND S_GREND  ; POORT VERGRENDELD  (SUB)
LD MALM_PAL1  ; ALARM PAL 1
ANDNOT SRESET  ; DK RESET BEDIEND (SUB)
ORLD
OUT MALMPAL1  ; PAL ALARM 1
; rung 2: ALM_PAL2 / IN ONDERSTAANDE GEVALLEN IS DE PAL OMLAAGGESTUURD / MAAR MELDT NIET LAAG
LD MI_STAP7  ; STAP 7 (SUB)
AND S_TIMER  ; STAPPENTIMER AFGELOPEN (SUB)
OR MI_STAP8  ; STAP 8 (SUB)
ANDNOT S_GREND  ; POORT VERGRENDELD  (SUB)
LD MALM_PAL2  ; ALARM PAL 2
ANDNOT SRESET  ; DK RESET BEDIEND (SUB)
ORLD
OUT MALMPAL2  ; PAL ALARM 2
; rung 3: ALM_OP1 / iN ONDERSTAANDE GEVALLEN MELDT DE OPEN SENSOR DAT DE / POORT OPEN IS TERWIJL DIT NIET KAN
LD MI_STAP8  ; STAP 8 (SUB)
AND S_OPEN  ; POORT OPEN (SUB)
LD MALM_OP1  ; ALARM OPEN SENSOR 1
ANDNOT SRESET  ; DK RESET BEDIEND (SUB)
ORLD
OUT MALMOP1  ; ALARM OPEN SENSOR 1
; rung 4: ALM_OP2 / IN ONDERSTAANDE GEVALLEN IS DE POORT GEOPEND MAAR DE / SENSOR OPEN MELDT DIT NIET
LD MI_STAP2  ; STAP 2 (SUB)
AND S_TIMER  ; STAPPENTIMER AFGELOPEN (SUB)
OR MI_STAP3  ; STAP 3 (SUB)
ANDNOT S_OPEN  ; POORT OPEN (SUB)
LD MALM_OP2  ; ALARM OPEN SENSOR 2
ANDNOT SRESET  ; DK RESET BEDIEND (SUB)
ORLD
OUT MALMOP2  ; ALARM OPEN SENSOR 2

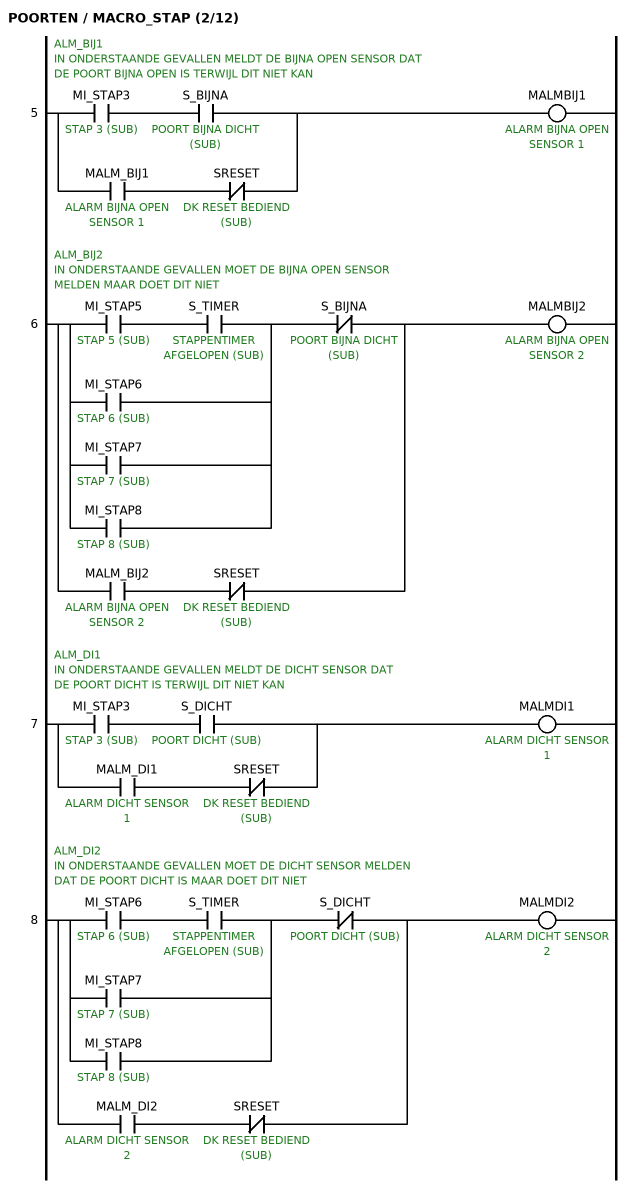
; rung 5: ALM_BIJ1 / IN ONDERSTAANDE GEVALLEN MELDT DE BIJNA OPEN SENSOR DAT / DE POORT BIJNA OPEN IS TERWIJL DIT NIET KAN
LD MI_STAP3  ; STAP 3 (SUB)
AND S_BIJNA  ; POORT BIJNA DICHT (SUB)
LD MALM_BIJ1  ; ALARM BIJNA OPEN SENSOR 1
ANDNOT SRESET  ; DK RESET BEDIEND (SUB)
ORLD
OUT MALMBIJ1  ; ALARM BIJNA OPEN SENSOR 1
; rung 6: ALM_BIJ2 / IN ONDERSTAANDE GEVALLEN MOET DE BIJNA OPEN SENSOR / MELDEN MAAR DOET DIT NIET
LD MI_STAP5  ; STAP 5 (SUB)
AND S_TIMER  ; STAPPENTIMER AFGELOPEN (SUB)
OR MI_STAP6  ; STAP 6 (SUB)
OR MI_STAP7  ; STAP 7 (SUB)
OR MI_STAP8  ; STAP 8 (SUB)
ANDNOT S_BIJNA  ; POORT BIJNA DICHT (SUB)
LD MALM_BIJ2  ; ALARM BIJNA OPEN SENSOR 2
ANDNOT SRESET  ; DK RESET BEDIEND (SUB)
ORLD
OUT MALMBIJ2  ; ALARM BIJNA OPEN SENSOR 2
; rung 7: ALM_DI1 / IN ONDERSTAANDE GEVALLEN MELDT DE DICHT SENSOR DAT / DE POORT DICHT IS TERWIJL DIT NIET KAN
LD MI_STAP3  ; STAP 3 (SUB)
AND S_DICHT  ; POORT DICHT (SUB)
LD MALM_DI1  ; ALARM DICHT SENSOR 1
ANDNOT SRESET  ; DK RESET BEDIEND (SUB)
ORLD
OUT MALMDI1  ; ALARM DICHT SENSOR 1
; rung 8: ALM_DI2 / IN ONDERSTAANDE GEVALLEN MOET DE DICHT SENSOR MELDEN / DAT DE POORT DICHT IS MAAR DOET DIT NIET
LD MI_STAP6  ; STAP 6 (SUB)
AND S_TIMER  ; STAPPENTIMER AFGELOPEN (SUB)
OR MI_STAP7  ; STAP 7 (SUB)
OR MI_STAP8  ; STAP 8 (SUB)
ANDNOT S_DICHT  ; POORT DICHT (SUB)
LD MALM_DI2  ; ALARM DICHT SENSOR 2
ANDNOT SRESET  ; DK RESET BEDIEND (SUB)
ORLD
OUT MALMDI2  ; ALARM DICHT SENSOR 2

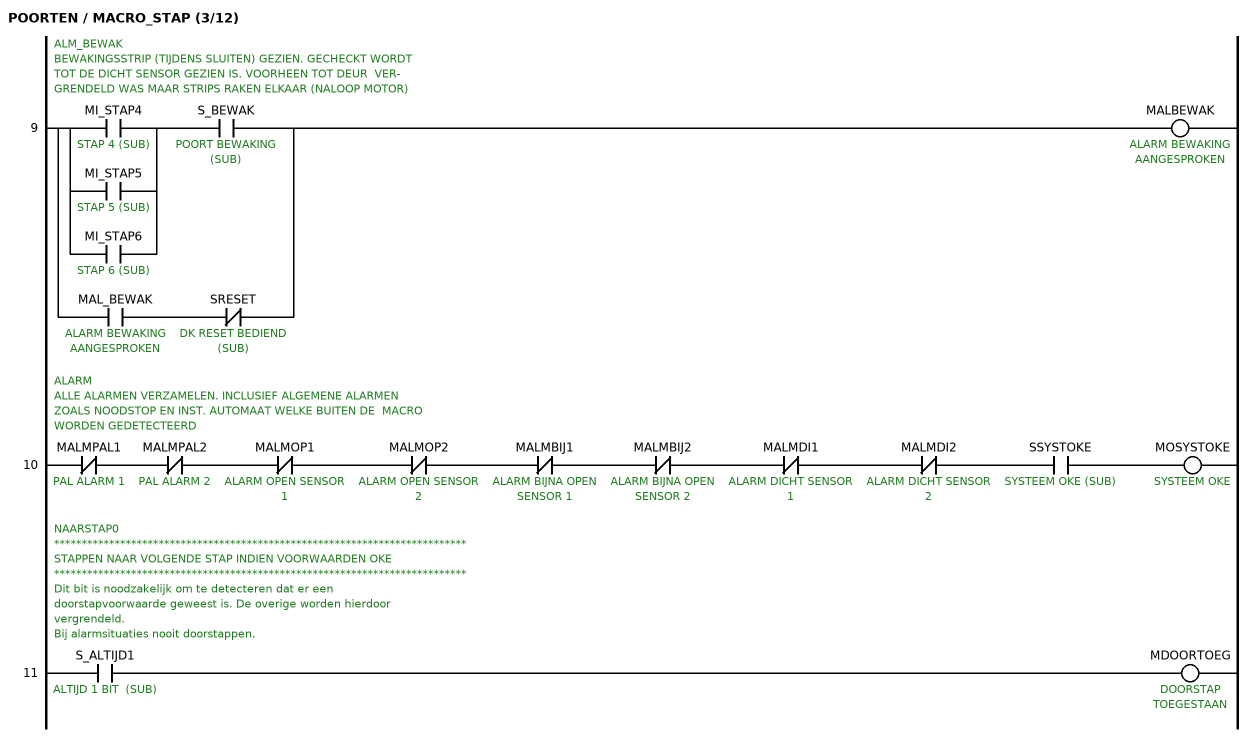
; rung 9: ALM_BEWAK / BEWAKINGSSTRIP (TIJDENS SLUITEN) GEZIEN. GECHECKT WORDT / TOT DE DICHT SENSOR GEZIEN IS. VOORHEEN TOT DEUR  VER- / GRENDELD WAS MAAR STRIPS RAKEN ELKAAR (NALOOP MOTOR)
LD MI_STAP4  ; STAP 4 (SUB)
OR MI_STAP5  ; STAP 5 (SUB)
OR MI_STAP6  ; STAP 6 (SUB)
AND S_BEWAK  ; POORT BEWAKING  (SUB)
LD MAL_BEWAK  ; ALARM BEWAKING AANGESPROKEN
ANDNOT SRESET  ; DK RESET BEDIEND (SUB)
ORLD
OUT MALBEWAK  ; ALARM BEWAKING AANGESPROKEN
; rung 10: ALARM / ALLE ALARMEN VERZAMELEN. INCLUSIEF ALGEMENE ALARMEN / ZOALS NOODSTOP EN INST. AUTOMAAT WELKE BUITEN DE  MACRO / WORDEN GEDETECTEERD
LDNOT MALMPAL1  ; PAL ALARM 1
ANDNOT MALMPAL2  ; PAL ALARM 2
ANDNOT MALMOP1  ; ALARM OPEN SENSOR 1
ANDNOT MALMOP2  ; ALARM OPEN SENSOR 2
ANDNOT MALMBIJ1  ; ALARM BIJNA OPEN SENSOR 1
ANDNOT MALMBIJ2  ; ALARM BIJNA OPEN SENSOR 2
ANDNOT MALMDI1  ; ALARM DICHT SENSOR 1
ANDNOT MALMDI2  ; ALARM DICHT SENSOR 2
AND SSYSTOKE  ; SYSTEEM OKE (SUB)
OUT MOSYSTOKE  ; SYSTEEM OKE
; rung 11: NAARSTAP0 / *************************************************************************** / STAPPEN NAAR VOLGENDE STAP INDIEN VOORWAARDEN OKE / *************************************************************************** / Dit bit is noodzakelijk om te detecteren dat er een / doorstapvoorwaarde geweest is. De overige worden hierdoor / vergrendeld. / Bij alarmsituaties nooit doorstappen.
LD S_ALTIJD1  ; ALTIJD 1 BIT  (SUB)
OUT MDOORTOEG  ; DOORSTAP TOEGESTAAN

